Staubli VAL3: decodeMsgBodyIO.pgx

public program decodeMsgBodyIO(RosSimpleMsg& x_rMsg, num& x_nMsgRecvState)
  local bool l_bFlag
begin
  // Copyright (c) 2016, Ocado Technology - Robotics Research Team
  //
  // Licensed under the Apache License, Version 2.0 (the "License");
  // you may not use this file except in compliance with the License.
  // You may obtain a copy of the License at
  //
  //     http://www.apache.org/licenses/LICENSE-2.0
  //
  // Unless required by applicable law or agreed to in writing, software
  // distributed under the License is distributed on an "AS IS" BASIS,
  // WITHOUT WARRANTIES OR CONDITIONS OF ANY KIND, either express or implied.
  // See the License for the specific language governing permissions and
  // limitations under the License.



  l_bFlag=false

  //switch x_rMsg.header.nMsgType
  //  case nStdMsgType["JOINT_TRAJ_PT"]
  //    call decTrajPt(l_bFlag)
  //  break
  //  case nStdMsgType["JOINT_TRAJ_PT_FULL"]
  //    call decTrajPtFull(l_bFlag)
  //  break
  //  case Staubli:MsgType.WRITE_SINGLE_IO
      call Staubli:decWriSingIOMsg(l_bFlag)
      logMsg("msgtype")
  //  break
  //  default
  //  break
  //endSwitch

  if (l_bFlag == true)
    // move on to state 4: push motion into buffer
    x_nMsgRecvState=nPushMotion
  else
    // error whilst decoding msg body...
    if (x_rMsg.header.nCommType==2)
      //switch x_rMsg.header.nMsgType
      //  case nStdMsgType["JOINT_TRAJ_PT"]
      //    rosTrajPtAck.header.nReplyCode=2
      //  break
      //  case nStdMsgType["JOINT_TRAJ_PT_FULL"]
      //    rosTrajPtFAck.header.nReplyCode=2
      //  break
      //  case Staubli:MsgType.WRITE_SINGLE_IO
          Staubli:writeSingIOAck.header.nReplyCode=SimpleMsg:ReplyCode.FAILURE
      //  break
      //  default
      //  break
      //endSwitch
      // jump to state 5: sendAck()
      x_nMsgRecvState=nAck
    else
      // reset state machine, since no ACK is required
      x_nMsgRecvState=nReset
    endIf
  endIf
end
